FUNCTION F_InLimits : BOOL
VAR_INPUT
    In        : LREAL;
    LowLimit  : LREAL;
    HighLimit : LREAL;
END_VAR

F_InLimits := (In >= LowLimit) AND (In <= HighLimit);

END_FUNCTION

(* stored: Version 1.1.0.1, ProductVersion 3.1.4024.12
   POU F_InLimits: Id {684d8a3f-78fd-42cb-9554-da2ecd9c9247}, SpecialFunc None *)
